// SIMATIC STEP 7 (V5.x) project firstLesson
// CPU: CPU 315-2 DP
// station: Hardware
// station: SIMATIC 300(1)
// station: P_ADR_BUS
// program: S7 Program(1)
// program: S7 Program(2)

ORGANIZATION_BLOCK OB 1
TITLE = "Main Program Sweep (Cycle)"
VERSION : 0.1
VAR_TEMP
  OB1_EV_CLASS : BYTE ;	//Bits 0-3 = 1 (Coming event), Bits 4-7 = 1 (Event class 1)
  OB1_SCAN_1 : BYTE ;	//1 (Cold restart scan 1 of OB 1), 3 (Scan 2-n of OB 1)
  OB1_PRIORITY : BYTE ;	//Priority of OB Execution
  OB1_OB_NUMBR : BYTE ;	//1 (Organization block 1, OB1)
  OB1_RESERVED_1 : BYTE ;	//Reserved for system
  OB1_RESERVED_2 : BYTE ;	//Reserved for system
  OB1_PREV_CYCLE : INT ;	//Cycle time of previous OB1 scan (milliseconds)
  OB1_MIN_CYCLE : INT ;	//Minimum cycle time of OB1 (milliseconds)
  OB1_MAX_CYCLE : INT ;	//Maximum cycle time of OB1 (milliseconds)
  OB1_DATE_TIME : DATE_AND_TIME ;	//Date and time OB1 started
END_VAR
BEGIN
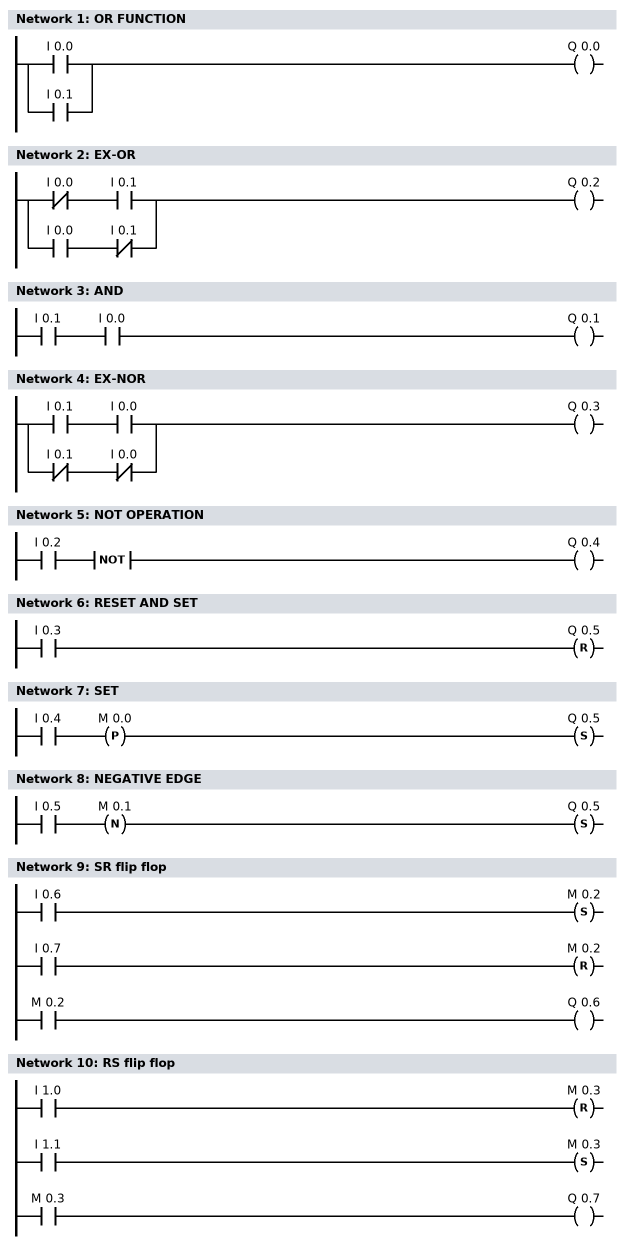
NETWORK
TITLE = OR FUNCTION
      O     I 0.0;
      O     I 0.1;
      =     Q 0.0;
NETWORK
TITLE = EX-OR
      AN    I 0.0;
      A     I 0.1;
      O;
      A     I 0.0;
      AN    I 0.1;
      =     Q 0.2;
NETWORK
TITLE = AND
      A     I 0.1;
      A     I 0.0;
      =     Q 0.1;
NETWORK
TITLE = EX-NOR
      A     I 0.1;
      A     I 0.0;
      O;
      AN    I 0.1;
      AN    I 0.0;
      =     Q 0.3;
NETWORK
TITLE = NOT OPERATION
      A     I 0.2;
      NOT;
      =     Q 0.4;
NETWORK
TITLE = RESET AND SET
      A     I 0.3;
      R     Q 0.5;
NETWORK
TITLE = SET
      A     I 0.4;
      FP    M 0.0;
      S     Q 0.5;
NETWORK
TITLE = NEGATIVE EDGE
      A     I 0.5;
      FN    M 0.1;
      S     Q 0.5;
NETWORK
TITLE = SR flip flop
      A     I 0.6;
      S     M 0.2;
      A     I 0.7;
      R     M 0.2;
      A     M 0.2;
      =     Q 0.6;
NETWORK
TITLE = RS flip flop
      A     I 1.0;
      R     M 0.3;
      A     I 1.1;
      S     M 0.3;
      A     M 0.3;
      =     Q 0.7;
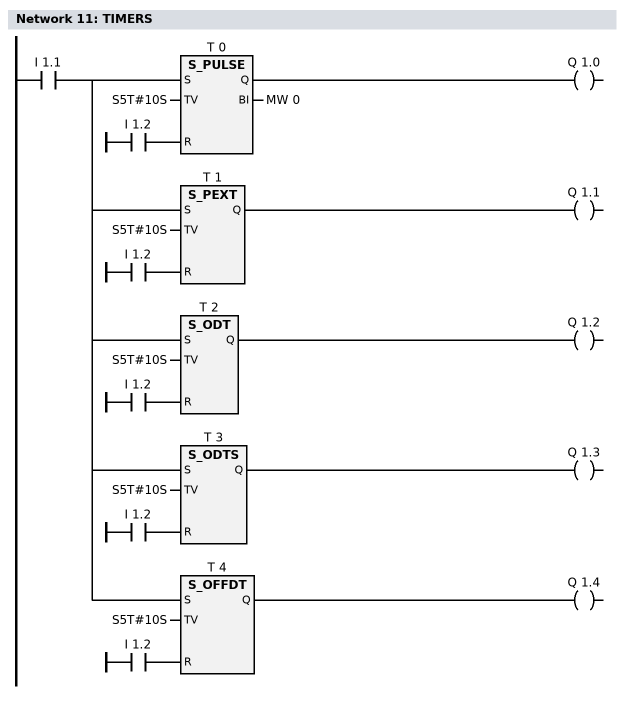
NETWORK
TITLE = TIMERS
      A     I 1.1;
      =     L 20.0;
      A     L 20.0;
      L     S5T#10S;
      SP    T 0;
      A     I 1.2;
      R     T 0;
      L     T 0;
      T     MW 0;
      NOP   0;
      A     T 0;
      =     Q 1.0;
      A     L 20.0;
      L     S5T#10S;
      SE    T 1;
      A     I 1.2;
      R     T 1;
      NOP   0;
      NOP   0;
      A     T 1;
      =     Q 1.1;
      A     L 20.0;
      L     S5T#10S;
      SD    T 2;
      A     I 1.2;
      R     T 2;
      NOP   0;
      NOP   0;
      A     T 2;
      =     Q 1.2;
      A     L 20.0;
      L     S5T#10S;
      SS    T 3;
      A     I 1.2;
      R     T 3;
      NOP   0;
      NOP   0;
      A     T 3;
      =     Q 1.3;
      A     L 20.0;
      L     S5T#10S;
      SF    T 4;
      A     I 1.2;
      R     T 4;
      NOP   0;
      NOP   0;
      A     T 4;
      =     Q 1.4;
END_ORGANIZATION_BLOCK

ORGANIZATION_BLOCK OB 2
VERSION : 0.1
VAR_TEMP
  Default: array [1..20] of byte;
END_VAR 
BEGIN
// (block stored without names or comments; labels and parameter names are numbered)
END_ORGANIZATION_BLOCK
